// TIA Portal V21 export
VAR_GLOBAL   // PLC tag table "Default tag table"
   System_Byte AT %MB1 : Byte;
   FirstScan AT %M1.0 : Bool;
   DiagStatusUpdate AT %M1.1 : Bool;
   AlwaysTRUE AT %M1.2 : Bool;
   AlwaysFALSE AT %M1.3 : Bool;
   Clock_Byte AT %MB0 : Byte;
   Clock_10Hz AT %M0.0 : Bool;
   Clock_5Hz AT %M0.1 : Bool;
   "Clock_2.5Hz" AT %M0.2 : Bool;
   Clock_2Hz AT %M0.3 : Bool;
   "Clock_1.25Hz" AT %M0.4 : Bool;
   Clock_1Hz AT %M0.5 : Bool;
   "Clock_0.625Hz" AT %M0.6 : Bool;
   "Clock_0.5Hz" AT %M0.7 : Bool;
   "+C0_K0.001" AT %I0.0 : Bool;   // Phase monitor OK
   "+C0_AUX/OK" AT %I0.1 : Bool;   // Auxiliary services protection OK
   "+C0_CAL/OK" AT %I0.2 : Bool;   // Heater protection OK
   "+C0_PE/OK" AT %I0.3 : Bool;   // Insulation monitor OK
   "+C0_Spare_101.4" AT %I0.4 : Bool;   // Spare
   "+C0_Spare_101.5" AT %I0.5 : Bool;   // Spare
   "+C0_Spare_101.6" AT %I0.6 : Bool;   // Spare
   "+C0_Spare_101.7" AT %I0.7 : Bool;   // Spare
   "+C0_S2.101" AT %I1.0 : Bool;   // Cabinet reset (power lines + emergencies)
   "+C0_S2.001" AT %I1.1 : Bool;   // Cabinet power lines deactivation
   "+C0_S2.002" AT %I1.2 : Bool;   // Acoustic warning stop
   "+C0_Spare_102.3" AT %I1.3 : Bool;   // Spare
   "+C0_IF5" AT %I1.4 : Bool;   // External machine interface 5
   "+C0_IF6" AT %I1.5 : Bool;   // External machine interface 6
   "+C0_IF7" AT %I1.6 : Bool;   // External machine interface 7
   "+C0_IF8" AT %I1.7 : Bool;   // External machine interface 8
   "+C0_F2.101" AT %I2.0 : Bool;   // 400V Power L1 protection OK
   "+C0_Q1.001" AT %I2.1 : Bool;   // Power L1 is active
   "+C0_1SE1" AT %I2.2 : Bool;   // Emergency stop 1 Z1 OK
   "+C0_1SE2" AT %I2.3 : Bool;   // Emergency stop 2 Z1 OK
   "+C0_F2.102" AT %I2.4 : Bool;   // 400V Power L2 protection OK
   "+C0_Q1.002" AT %I2.5 : Bool;   // Power L2 is active
   "+C0_2SE1" AT %I2.6 : Bool;   // Emergency stop 1 Z2 OK
   "+C0_2SE2" AT %I2.7 : Bool;   // Emergency stop 2 Z2 OK
   "+C0_F2.103" AT %I3.0 : Bool;   // 400V Power L3 protection OK
   "+C0_Q1.003" AT %I3.1 : Bool;   // Power L3 is active
   "+C0_3SE1" AT %I3.2 : Bool;   // Emergency stop 1 Z3 OK
   "+C0_3SE2" AT %I3.3 : Bool;   // Emergency stop 2 Z3 OK
   "+C0_F2.104" AT %I3.4 : Bool;   // 400V Power L4 protection OK
   "+C0_Q1.004" AT %I3.5 : Bool;   // Power L4 is active
   "+C0_4SE1" AT %I3.6 : Bool;   // Emergency stop 1 Z4 OK
   "+C0_4SE2" AT %I3.7 : Bool;   // Emergency stop 2 Z4 OK
   "+C0_F2.105" AT %I4.0 : Bool;   // 400V Power L5 protection OK
   "+C0_Q1.005" AT %I4.1 : Bool;   // Power L5 is active
   "+C0_5SE1" AT %I4.2 : Bool;   // Emergency stop 1 Z5 OK
   "+C0_5SE2" AT %I4.3 : Bool;   // Emergency stop 2 Z5 OK
   "+C0_F2.106" AT %I4.4 : Bool;   // 400V Power L6 protection OK
   "+C0_Q1.006" AT %I4.5 : Bool;   // Power L6 is active
   "+C0_6SE1" AT %I4.6 : Bool;   // Emergency stop 1 Z6 OK
   "+C0_6SE2" AT %I4.7 : Bool;   // Emergency stop 2 Z6 OK
   "+C0_Spare_106.1" AT %I5.1 : Bool;   // Spare
   "+C0_7SE1" AT %I5.2 : Bool;   // Emergency stop 1 Z7 OK
   "+C0_7SE2" AT %I5.3 : Bool;   // Emergency stop 2 Z7 OK
   "+C0_Spare_106.4" AT %I5.4 : Bool;   // Spare
   "+C0_Spare_106.5" AT %I5.5 : Bool;   // Spare
   "+C0_8SE1" AT %I5.6 : Bool;   // Emergency stop 1 Z8 OK
   "+C0_8SE2" AT %I5.7 : Bool;   // Emergency stop 2 Z8 OK
   "+C0_F0.199 -F2.199" AT %I6.0 : Bool;   // Wrapping machine protection OK
   "+C0_ENF1" AT %I6.1 : Bool;   // Wrapping machine is ready
   "+C0_ENF2" AT %I6.2 : Bool;   // Wrapping machine entry consent
   "+C0_ENF3" AT %I6.3 : Bool;   // Wrapping machine completed process
   "+C0_Spare_107.4" AT %I6.4 : Bool;   // Spare
   "+C0_Spare_107.5" AT %I6.5 : Bool;   // Spare
   "+C0_Spare_107.6" AT %I6.6 : Bool;   // Spare
   "+C0_Spare_107.7" AT %I6.7 : Bool;   // Spare
   "+C0_F0.190+" AT %I7.0 : Bool;   // Fast doors protection OK
   "+C0_1PR1" AT %I7.1 : Bool;   // Fast door 1 is open
   "+C0_1PR2" AT %I7.2 : Bool;   // Fast door 1 is closed
   "+C0_2PR1" AT %I7.3 : Bool;   // Fast door 2 is open
   "+C0_2PR2" AT %I7.4 : Bool;   // Fast door 2 is closed
   "+C0_3PR1" AT %I7.5 : Bool;   // Fast door 3 is open
   "+C0_3PR2" AT %I7.6 : Bool;   // Fast door 3 is closed
   "+C0_Spare_108.7" AT %I7.7 : Bool;   // Spare
   "+C0_Buzzer" AT %Q0.0 : Bool;   // Beacon buzzer
   "+C0_Beacon_Green" AT %Q0.1 : Bool;   // Beacon green lamp
   "+C0_Beacon_Red" AT %Q0.2 : Bool;   // Beacon red lamp
   "+C0_Spare_151.3" AT %Q0.3 : Bool;   // Spare
   "+C0_PEM" AT %Q0.4 : Bool;   // Cabinet emergency stop is active
   "+C0_RE" AT %Q0.5 : Bool;   // Cabinet power lines are active
   "+C0_Spare_151.6" AT %Q0.6 : Bool;   // Spare
   "+C0_Spare_151.7" AT %Q0.7 : Bool;   // Spare
   "+C0_K1.007" AT %Q1.0 : Bool;   // External machine interface 1
   "+C0_K1.008" AT %Q1.1 : Bool;   // External machine interface 2
   "+C0_K1.009" AT %Q1.2 : Bool;   // External machine interface 3
   "+C0_K1.010" AT %Q1.3 : Bool;   // External machine interface 4
   "+C0_Spare_152.4" AT %Q1.4 : Bool;   // Spare
   "+C0_Spare_152.5" AT %Q1.5 : Bool;   // Spare
   "+C0_Spare_152.6" AT %Q1.6 : Bool;   // Spare
   "+C0_Spare_152.7" AT %Q1.7 : Bool;   // Spare
   "+C0_K1.001" AT %Q2.0 : Bool;   // 400V Power L1 activation
   "+C0_K1.002" AT %Q2.1 : Bool;   // 400V Power L2 activation
   "+C0_K1.003" AT %Q2.2 : Bool;   // 400V Power L3 activation
   "+C0_K1.004" AT %Q2.3 : Bool;   // 400V Power L4 activation
   "+C0_K1.005" AT %Q2.4 : Bool;   // 400V Power L5 activation
   "+C0_K1.006" AT %Q2.5 : Bool;   // 400V Power L6 activation
   "+C0_Spare_153.6" AT %Q2.6 : Bool;   // Spare
   "+C0_Spare_153.7" AT %Q2.7 : Bool;   // Spare
   "+C0_K1.020" AT %Q3.0 : Bool;   // Wrapping machine exit request
   "+C0_Spare_154.1" AT %Q3.1 : Bool;   // Spare
   "+C0_K1.030" AT %Q3.2 : Bool;   // Open fast door 1
   "+C0_K1.031" AT %Q3.3 : Bool;   // Close fast door 1
   "+C0_K1.032" AT %Q3.4 : Bool;   // Open fast door 2
   "+C0_K1.033" AT %Q3.5 : Bool;   // Close fast door 2
   "+C0_K1.035" AT %Q3.7 : Bool;   // Close fast door 3
   "+C0_S1.001_1" AT %I100.0 : Bool;   // Cabinet emergency stop ch1
   "+C0_Spare_201.1" AT %I100.1 : Bool;   // Spare
   "+C0_Spare_201.2" AT %I100.2 : Bool;   // Spare
   "+C0_Spare_201.3" AT %I100.3 : Bool;   // Spare
   "+C0_S1.001_2" AT %I100.4 : Bool;   // Cabinet emergency stop ch2
   "+C0_Spare_201.5" AT %I100.5 : Bool;   // Spare
   "+C0_Spare_201.6" AT %I100.6 : Bool;   // Spare
   "+C0_Spare_201.7" AT %I100.7 : Bool;   // Spare
   "+C0_1EM1" AT %I107.0 : Bool;   // Emergency stop Z1 ch1
   "+C0_2EM1" AT %I107.1 : Bool;   // Emergency stop Z2 ch1
   "+C0_K4.011-111-012-112" AT %I107.2 : Bool;   // Safety Z1 relays feedback
   "+C0_Spare_202.3" AT %I107.3 : Bool;   // Spare
   "+C0_1EM2" AT %I107.4 : Bool;   // Emergency stop Z1 ch2
   "+C0_2EM2" AT %I107.5 : Bool;   // Emergency stop Z2 ch2
   "+C0_K4.021-121-022-122" AT %I107.6 : Bool;   // Safety Z2 relays feedback
   "+C0_Spare_202.7" AT %I107.7 : Bool;   // Sapre
   "+C0_3EM1" AT %I114.0 : Bool;   // Emergency stop Z3 ch1
   "+C0_4EM1" AT %I114.1 : Bool;   // Emergency stop Z4 ch1
   "+C0_K4.031-131-032-132" AT %I114.2 : Bool;   // Safety Z3 relays feedback
   "+C0_Spare_203.3" AT %I114.3 : Bool;   // Spare
   "+C0_3EM2" AT %I114.4 : Bool;   // Emergency stop Z3 ch2
   "+C0_4EM2" AT %I114.5 : Bool;   // Emergency stop Z4 ch2
   "+C0_K4.041-141-042-142" AT %I114.6 : Bool;   // Safety Z4 relays feedback
   "+C0_Spare_203.7" AT %I114.7 : Bool;   // Spare
   "+C0_5EM1" AT %I121.0 : Bool;   // Emergency stop Z5 ch1
   "+C0_6EM1" AT %I121.1 : Bool;   // Emergency stop Z6 ch1
   "+C0_K4.051-151-052-152" AT %I121.2 : Bool;   // Safety Z5 relays feedback
   "+C0_Spare_204.3" AT %I121.3 : Bool;   // Spare
   "+C0_5EM2" AT %I121.4 : Bool;   // Emergency stop Z5 ch2
   "+C0_6EM2" AT %I121.5 : Bool;   // Emergency stop Z6 ch2
   "+C0_K4.061-161-062-162" AT %I121.6 : Bool;   // Safety Z6 relays feedback
   "+C0_Spare_204.7" AT %I121.7 : Bool;   // Spare
   "+C0_7EM1" AT %I128.0 : Bool;   // Emergency stop Z7 ch1
   "+C0_8EM1" AT %I128.1 : Bool;   // Emergency stop Z8 ch1
   "+C0_K4.071-171-072-172" AT %I128.2 : Bool;   // Safety Z7 relays feedback
   "+C0_Spare_205.3" AT %I128.3 : Bool;   // Spare
   "+C0_7EM2" AT %I128.4 : Bool;   // Emergency stop Z7 ch2
   "+C0_8EM2" AT %I128.5 : Bool;   // Emergency stop Z8 ch2
   "+C0_K4.081-181-082-182" AT %I128.6 : Bool;   // Safety Z8 relays feedback
   "+C0_Spare_205.7" AT %I128.7 : Bool;   // Spare
   "+C0_K4.011-111" AT %Q200.0 : Bool;   // Safety Z1 ch1 relay activation
   "+C0_K4.012-112" AT %Q200.1 : Bool;   // Safety Z1 ch2 relay activation
   "+C0_K4.021-121" AT %Q200.2 : Bool;   // Safety Z2 ch1 relay activation
   "+C0_K4.022-122" AT %Q200.3 : Bool;   // Safety Z2 ch2 relay activation
   "+C0_K4.031-131" AT %Q200.4 : Bool;   // Safety Z3 ch1 relay activation
   "+C0_K4.032-132" AT %Q200.5 : Bool;   // Safety Z3 ch2 relay activation
   "+C0_K4.041-141" AT %Q200.6 : Bool;   // Safety Z4 ch1 relay activation
   "+C0_K4.042-142" AT %Q200.7 : Bool;   // Safety Z4 ch2 relay activation
   "+C0_K4.051-151" AT %Q206.0 : Bool;   // Safety Z5 ch1 relay activation
   "+C0_K4.052-152" AT %Q206.1 : Bool;   // Safety Z5 ch2 relay activation
   "+C0_K4.061-161" AT %Q206.2 : Bool;   // Safety Z6 ch1 relay activation
   "+C0_K4.062-162" AT %Q206.3 : Bool;   // Safety Z6 ch2 relay activation
   "+C0_K4.071-171" AT %Q206.4 : Bool;   // Safety Z7 ch1 relay activation
   "+C0_K4.072-172" AT %Q206.5 : Bool;   // Safety Z7 ch2 relay activation
   "+C0_K4.081-181" AT %Q206.6 : Bool;   // Safety Z8 ch1 relay activation
   "+C0_K4.082-182" AT %Q206.7 : Bool;   // Safety Z8 ch2 relay activation
   "+C0_A0.101" AT %IB0 : Byte;
   "+C0_A0.102" AT %IB1 : Byte;
   "+C0_A0.103" AT %IB2 : Byte;
   "+C0_A0.104" AT %IB3 : Byte;
   "+C0_A0.105" AT %IB4 : Byte;
   "+C0_A0.106" AT %IB5 : Byte;
   "+C0_A0.107" AT %IB6 : Byte;
   "+C0_A0.108" AT %IB7 : Byte;
   "+C0_Spare_106.0" AT %I5.0 : Bool;   // Spare
   "+C0_K1.034" AT %Q3.6 : Bool;   // Open fast door 3
   RONDI_PEM_20260514 AT %M650.0 : Bool;   // VARIABLE DE PUESTA EN MARCHA
   MOTOR_ON AT %M650.1 : Bool;
END_VAR
